INTERFACE I_Module

METHOD Disable
END_METHOD

METHOD Enable
END_METHOD

END_INTERFACE

(* stored: Version 1.1.0.1, ProductVersion 3.1.4024.11
   Itf I_Module: Id {871b2712-10c1-4ee2-ac36-2459f4f56cfc}
   Method Disable: Id {0ad36714-3107-476d-b6f5-b053eac7356c}
   Method Enable: Id {ed3b2922-ceb7-48b3-a4f5-fe6a4cea96a8} *)
